// TwinCAT 3 PLC project PLC
// ProgramVersion: 3.1.4026.14
// CompilerDefines: VISU_USEPROPERTYINFO
// libraries:
//   SPT Base Types, * (Beckhoff Automation LLC)
//   SPT Components, * (Beckhoff Automation LLC)
//   SPT Diagnostic, * (Beckhoff Automation LLC)
//   SPT EtherCat, * (Beckhoff Automation LLC)
//   SPT Event Logger, * (Beckhoff Automation LLC)
//   SPT Kinematics, * (Beckhoff Automation LLC)
//   SPT Motion Control, * (Beckhoff Automation LLC)
//   SPT NCI, * (Beckhoff Automation LLC)
//   SPT Utilities, * (Beckhoff Automation LLC)
//   SPT Vision, * (Beckhoff Automation LLC)
//   SPT XTS, * (Beckhoff Automation LLC)
//   Tc2_Standard, * (Beckhoff Automation GmbH)
//   Tc2_System, * (Beckhoff Automation GmbH)
//   Tc3_EventLogger, * (Beckhoff Automation GmbH)
//   Tc3_PackML_V2, * (Beckhoff Automation GmbH)
// project tree:
//   / GlobalTextList.TcGTLO (not stored), PlcTask.TcTTO (not stored), VisualizationManager.TcVMO (not stored)
//   POUs/ Machine.TcPOU (not stored), MAIN.TcPOU
//   VISUs/ Visualization.TcVIS
// real-time tasks:
//   TASK PlcTask: cycle T#10ms, priority 20, ADS port 350

// ---- POUs/MAIN.TcPOU
PROGRAM MAIN
VAR
	Machine : Machine := (Name := 'Machine');
END_VAR

(*All sample code provided by Beckhoff Automation LLC are for illustrative purposes only and are provided “as is” and without any warranties, express or implied. Actual implementations in applications will vary significantly. Beckhoff Automation LLC shall have no liability for, and does not waive any rights in relation to, any code samples that it provides or the use of such code samples for any purpose.*)

(*
	This example is the smallest possible implementation of the the framework. 
	By calling the CyclicLogic of Machine everything inside the framework that is needed to control the statemachine and log the existing events is being processed.
	
	The HMIPermissions method is required to allow the Visu to control the state machine through the PackMLBaseModule_HMI structure.
	
	All libraries in this project are pinned at V3.9.x
	While only the SPT Base Types library is used, the others are provided for your convenience.
	
*)

Machine.CyclicLogic();

END_PROGRAM

// ---- VISUs/Visualization.TcVIS
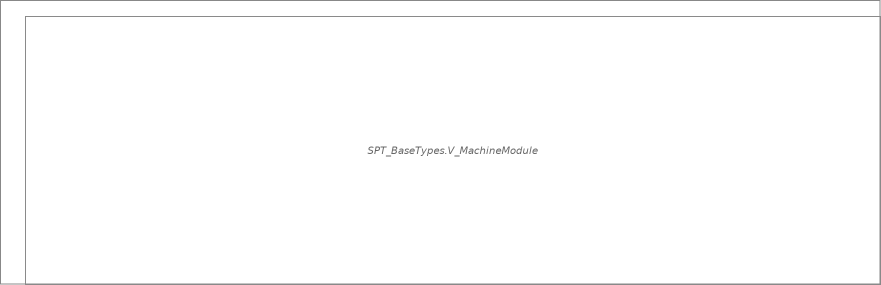
VISUALIZATION Visualization  // 881x285
    Frame (25,16 856x269)
        shows SPT_BaseTypes.V_MachineModule(HMI := MAIN.Machine.PackMLBaseModule_HMI)
END_VISUALIZATION
